// TIA Portal V16 export
// export: Created 2025-05-30T16:35:57.2781598Z, ExportSetting WithDefaults, DisplayName Totally Integrated Automation Portal, DisplayVersion V16, DisplayName TIA Portal Version Control Interface, DisplayVersion V16, DisplayName TIA Portal Openness, DisplayVersion V16, DisplayName STEP 7 Professional, DisplayVersion V16, DisplayName STEP 7 Safety, DisplayVersion V16, DisplayName WinCC Advanced, DisplayVersion V16
FUNCTION_BLOCK "Programma 1 - Test"   // FB12, GRAPH
VERSION : 0.1
// stored: AcknowledgeErrorsRequired true, AutoNumber true, CreateMinimizedDB false, IsIECCheckEnabled false, LanguageInNetworks LAD, LockOperatingMode false, PermanentILProcessingInMANMode false, SkipSteps false, UDAEnableTagReadback false, WithAlarmHandling true
   VAR_INPUT
      OFF_SQ { ExternalAccessible := 'False'; ExternalVisible := 'False'; ExternalWritable := 'False'} : Bool := false;   // Turn sequence off
      INIT_SQ { ExternalAccessible := 'False'; ExternalVisible := 'False'; ExternalWritable := 'False'} : Bool := false;   // Set sequence to initial state
      ACK_EF { ExternalAccessible := 'False'; ExternalVisible := 'False'; ExternalWritable := 'False'} : Bool := false;   // Acknowledge all errors and faults
      S_PREV { ExternalAccessible := 'False'; ExternalVisible := 'False'; ExternalWritable := 'False'} : Bool := false;   // Output previous step in parameter S_NO
      S_NEXT { ExternalAccessible := 'False'; ExternalVisible := 'False'; ExternalWritable := 'False'} : Bool := false;   // Indicate next step in parameter S_NO
      SW_AUTO { ExternalAccessible := 'False'; ExternalVisible := 'False'; ExternalWritable := 'False'} : Bool := false;   // Automatic mode
      SW_TAP { ExternalAccessible := 'False'; ExternalVisible := 'False'; ExternalWritable := 'False'} : Bool := false;   // Semiautomatic/switch with transition
      SW_TOP { ExternalAccessible := 'False'; ExternalVisible := 'False'; ExternalWritable := 'False'} : Bool := false;   // Semiautomatic/ignore transition
      SW_MAN { ExternalAccessible := 'False'; ExternalVisible := 'False'; ExternalWritable := 'False'} : Bool := false;   // Manual mode
      S_SEL { ExternalAccessible := 'False'; ExternalVisible := 'False'; ExternalWritable := 'False'} : Int := 0;   // Select step to be output to S_NO
      S_ON { ExternalAccessible := 'False'; ExternalVisible := 'False'; ExternalWritable := 'False'} : Bool := false;   // Activate step indicated in S_NO
      S_OFF { ExternalAccessible := 'False'; ExternalVisible := 'False'; ExternalWritable := 'False'} : Bool := false;   // Deactivate step indicated S_NO
      T_PUSH { ExternalAccessible := 'False'; ExternalVisible := 'False'; ExternalWritable := 'False'} : Bool := false;   // Enable transition to switch in semi automatic mode
      "Confimation Position 1" : Bool;
      "Confirmation Position 2" : Bool;
      "Products more than zero" : Bool;
      "Products zero" : Bool;
      "Timer 1" : Time;
   END_VAR
   VAR_OUTPUT
      S_NO { ExternalAccessible := 'False'; ExternalVisible := 'False'; ExternalWritable := 'False'} : Int := 0;   // Step number
      S_MORE { ExternalAccessible := 'False'; ExternalVisible := 'False'; ExternalWritable := 'False'} : Bool := false;   // More steps are available and can be shown in S_NO
      S_ACTIVE { ExternalAccessible := 'False'; ExternalVisible := 'False'; ExternalWritable := 'False'} : Bool := false;   // Step indicated in S_NO is active
      ERR_FLT { ExternalAccessible := 'False'; ExternalVisible := 'False'; ExternalWritable := 'False'} : Bool := false;   // Interlock or supervision group error
      AUTO_ON { ExternalAccessible := 'False'; ExternalVisible := 'False'; ExternalWritable := 'False'} : Bool := false;   // Automatic mode is active
      TAP_ON { ExternalAccessible := 'False'; ExternalVisible := 'False'; ExternalWritable := 'False'} : Bool := false;   // Semiautomatic mode/step with transition enabled
      TOP_ON { ExternalAccessible := 'False'; ExternalVisible := 'False'; ExternalWritable := 'False'} : Bool := false;   // Semiautomatic mode/ignore transition enabled
      MAN_ON { ExternalAccessible := 'False'; ExternalVisible := 'False'; ExternalWritable := 'False'} : Bool := false;   // Manual mode is active
      "Move Position 1" : Bool;
      "Move Position 2" : Bool;
   END_VAR
   VAR DB_SPECIFIC
      S_DISPLAY { ExternalAccessible := 'False'; ExternalVisible := 'False'; ExternalWritable := 'False'} : Int;   // Internal display of output parameter S_NO
      S_SEL_OLD { ExternalAccessible := 'False'; ExternalVisible := 'False'; ExternalWritable := 'False'} : Int;   // Previous value in S_SEL
      S_DISPIDX { ExternalAccessible := 'False'; ExternalVisible := 'False'; ExternalWritable := 'False'} : Byte;   // Index of the step in S_NO
      T_DISPIDX { ExternalAccessible := 'False'; ExternalVisible := 'False'; ExternalWritable := 'False'} : Byte;   // Index of the transition displayed in T_NO
      MOP { ExternalAccessible := 'False'; ExternalVisible := 'False'; ExternalWritable := 'False'} : Struct   // Mode
         AUTO { ExternalAccessible := 'False'; ExternalVisible := 'False'; ExternalWritable := 'False'} : Bool := true;   // Status: automatic mode
         MAN { ExternalAccessible := 'False'; ExternalVisible := 'False'; ExternalWritable := 'False'} : Bool := false;   // Status: manual mode
         TAP { ExternalAccessible := 'False'; ExternalVisible := 'False'; ExternalWritable := 'False'} : Bool := false;   // Status: semi automatic/switch with transition
         TOP { ExternalAccessible := 'False'; ExternalVisible := 'False'; ExternalWritable := 'False'} : Bool := false;   // Status: semi automatic/ignore transition
         ACK_S { ExternalAccessible := 'False'; ExternalVisible := 'False'; ExternalWritable := 'False'} : Bool := false;   // Request: acknowledge step at parameter S_NO
         REG_S { ExternalAccessible := 'False'; ExternalVisible := 'False'; ExternalWritable := 'False'} : Bool := false;   // Request: register step indicated in S_NO
         T_PREV { ExternalAccessible := 'False'; ExternalVisible := 'False'; ExternalWritable := 'False'} : Bool := false;   // Request: output previous valid transition in T_NO
         T_NEXT { ExternalAccessible := 'False'; ExternalVisible := 'False'; ExternalWritable := 'False'} : Bool := false;   // Request: output next valid transition in T_NO
         LOCK { ExternalAccessible := 'False'; ExternalVisible := 'False'; ExternalWritable := 'False'} : Bool := true;   // Status: interlocks activated
         SUP { ExternalAccessible := 'False'; ExternalVisible := 'False'; ExternalWritable := 'False'} : Bool := true;   // Status: supervisions activated
         ACKREQ { ExternalAccessible := 'False'; ExternalVisible := 'False'; ExternalWritable := 'False'} : Bool := true;   // Status: acknowledgment required
         SSKIP { ExternalAccessible := 'False'; ExternalVisible := 'False'; ExternalWritable := 'False'} : Bool := false;   // Status: "Skip steps" enabled
         OFF { ExternalAccessible := 'False'; ExternalVisible := 'False'; ExternalWritable := 'False'} : Bool := false;   // Request: deactivate all steps
         INIT { ExternalAccessible := 'False'; ExternalVisible := 'False'; ExternalWritable := 'False'} : Bool := true;   // Request: set sequence to initial state
         HALT { ExternalAccessible := 'False'; ExternalVisible := 'False'; ExternalWritable := 'False'} : Bool := false;   // Status: sequence halted
         TMS_HALT { ExternalAccessible := 'False'; ExternalVisible := 'False'; ExternalWritable := 'False'} : Bool := false;   // Status: all internal timers held
         OPS_ZERO { ExternalAccessible := 'False'; ExternalVisible := 'False'; ExternalWritable := 'False'} : Bool := false;   // Status: set all operands processed with N, L, D instructions to 0
         SACT_DISP { ExternalAccessible := 'False'; ExternalVisible := 'False'; ExternalWritable := 'False'} : Bool := true;   // Status: display active steps only
         SEF_DISP { ExternalAccessible := 'False'; ExternalVisible := 'False'; ExternalWritable := 'False'} : Bool := false;   // Status: display only steps with errors and disrupted steps
         SALL_DISP { ExternalAccessible := 'False'; ExternalVisible := 'False'; ExternalWritable := 'False'} : Bool := false;   // Status: display all steps
         S_PREV { ExternalAccessible := 'False'; ExternalVisible := 'False'; ExternalWritable := 'False'} : Bool := false;   // Request: output previous step to S_NO
         S_NEXT { ExternalAccessible := 'False'; ExternalVisible := 'False'; ExternalWritable := 'False'} : Bool := false;   // Request: Output next step at S_NO parameter
         S_SELOK { ExternalAccessible := 'False'; ExternalVisible := 'False'; ExternalWritable := 'False'} : Bool := false;   // Request: output step number from S_SEL to S_NO
         S_ON { ExternalAccessible := 'False'; ExternalVisible := 'False'; ExternalWritable := 'False'} : Bool := false;   // Request: activate step indicated in S_NO
         S_OFF { ExternalAccessible := 'False'; ExternalVisible := 'False'; ExternalWritable := 'False'} : Bool := false;   // Request: deactivate step at parameter S_NO
         T_PUSH { ExternalAccessible := 'False'; ExternalVisible := 'False'; ExternalWritable := 'False'} : Bool := false;   // Request: transition switching enabled
         REG { ExternalAccessible := 'False'; ExternalVisible := 'False'; ExternalWritable := 'False'} : Bool := false;   // Request: register all interlock and supervision errors
         ACK { ExternalAccessible := 'False'; ExternalVisible := 'False'; ExternalWritable := 'False'} : Bool := false;   // Request: acknowledge all interlock and supervision errors
         IL_PERM { ExternalAccessible := 'False'; ExternalVisible := 'False'; ExternalWritable := 'False'} : Bool := false;   // Status: permanent processing of all interlocks
         T_PERM { ExternalAccessible := 'False'; ExternalVisible := 'False'; ExternalWritable := 'False'} : Bool := false;   // Status: permanent processing of all transitions
         ILP_MAN { ExternalAccessible := 'False'; ExternalVisible := 'False'; ExternalWritable := 'False'} : Bool := false;   // Status: permanent processing of all interlocks in manual mode
      END_STRUCT;
      TICKS { ExternalAccessible := 'False'; ExternalVisible := 'False'; ExternalWritable := 'False'} : Struct   // Clock speeds
         DELTA { ExternalAccessible := 'False'; ExternalVisible := 'False'; ExternalWritable := 'False'} : Time := T#0ms;   // Time difference between cycles
         OLD { ExternalAccessible := 'False'; ExternalVisible := 'False'; ExternalWritable := 'False'} : Time := T#0ms;   // 10 ms clock counter value in last cycle
         NEW { ExternalAccessible := 'False'; ExternalVisible := 'False'; ExternalWritable := 'False'} : Time := T#0ms;   // 10 ms clock counter value in this cycle
      END_STRUCT;
      SQ_FLAGS { ExternalAccessible := 'False'; ExternalVisible := 'False'; ExternalWritable := 'False'} : Struct   // Sequence bit memory
         ERR_FLT { ExternalAccessible := 'False'; ExternalVisible := 'False'; ExternalWritable := 'False'} : Bool := false;   // Interlock and supervision group error
         ERROR { ExternalAccessible := 'False'; ExternalVisible := 'False'; ExternalWritable := 'False'} : Bool := false;   // Interlock group error
         FAULT { ExternalAccessible := 'False'; ExternalVisible := 'False'; ExternalWritable := 'False'} : Bool := false;   // Supervision group error
         RT_FAIL { ExternalAccessible := 'False'; ExternalVisible := 'False'; ExternalWritable := 'False'} : Bool := false;   // Runtime error
         NO_SNO { ExternalAccessible := 'False'; ExternalVisible := 'False'; ExternalWritable := 'False'} : Bool := false;   // Requested step number not found
         NF_OFL { ExternalAccessible := 'False'; ExternalVisible := 'False'; ExternalWritable := 'False'} : Bool := false;   // Overflow: too many ON or OFF requests
         SA_OFL { ExternalAccessible := 'False'; ExternalVisible := 'False'; ExternalWritable := 'False'} : Bool := false;   // Overflow: too many steps active
         TV_OFL { ExternalAccessible := 'False'; ExternalVisible := 'False'; ExternalWritable := 'False'} : Bool := false;   // Overflow: too many valid transitions
         MSG_OFL { ExternalAccessible := 'False'; ExternalVisible := 'False'; ExternalWritable := 'False'} : Bool := false;   // Overflow: not enough system resources for ALARM_S
         NO_SWI { ExternalAccessible := 'False'; ExternalVisible := 'False'; ExternalWritable := 'False'} : Bool := false;   // Do not switch in this cycle
         CYC_OP { ExternalAccessible := 'False'; ExternalVisible := 'False'; ExternalWritable := 'False'} : Bool := false;   // Cyclic execution of the sequence after initialization
         AS_MSG { ExternalAccessible := 'False'; ExternalVisible := 'False'; ExternalWritable := 'False'} : Bool := true;   // Alarms during runtime enabled or disabled by instruction
         AS_SEND { ExternalAccessible := 'False'; ExternalVisible := 'False'; ExternalWritable := 'False'} : Bool := false;   // Send alarms from WR_USMSG or only enter in diagnostics buffer
         SQ_BUSY { ExternalAccessible := 'False'; ExternalVisible := 'False'; ExternalWritable := 'False'} : Bool := false;   // Internal edge memory bit for sequence processing
         SA_BUSY { ExternalAccessible := 'False'; ExternalVisible := 'False'; ExternalWritable := 'False'} : Bool := false;   // Internal edge memory bit for sequence processing
         AS_SIG { ExternalAccessible := 'False'; ExternalVisible := 'False'; ExternalWritable := 'False'} : Bool := false;   // Edge memory bit for alarms from Alarm_S and Alarm_SQ
      END_STRUCT;
   END_VAR
BEGIN
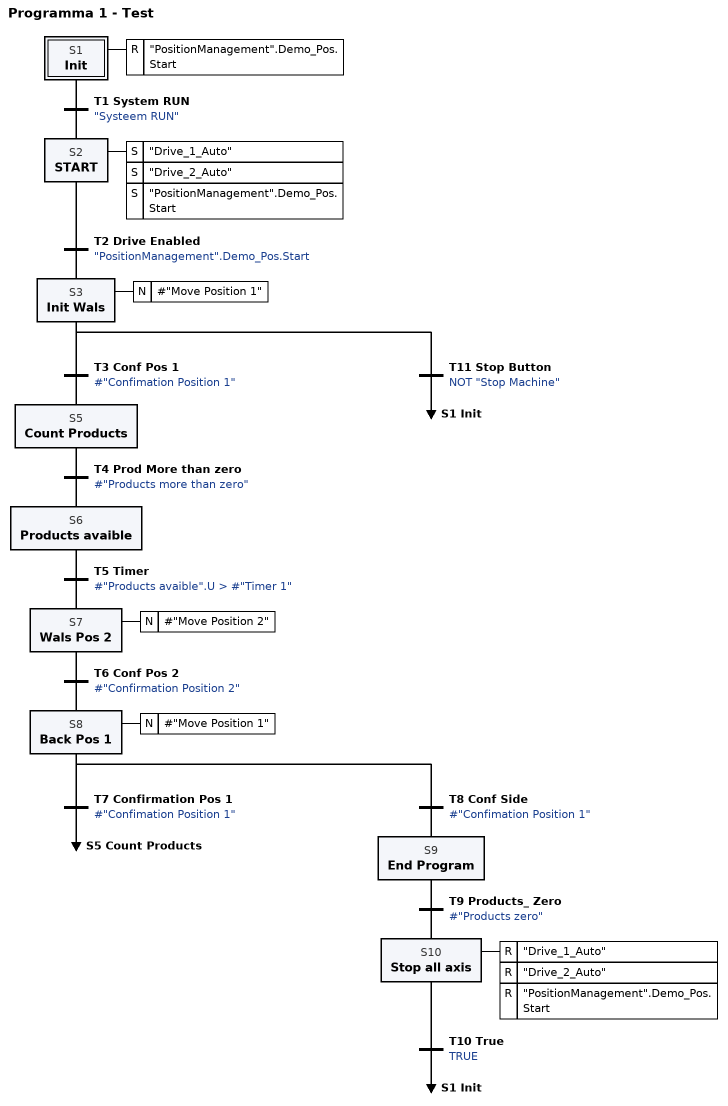
   // sequencer 1: SFC Program
   INITIAL_STEP Init:   // S1
              R    "PositionManagement".Demo_Pos.Start
   END_STEP
   TRANSITION "System RUN" FROM Init TO START   // T1
      := "Systeem RUN";
   END_TRANSITION
   STEP START:   // S2
      // Set Ouputs
              S    "Drive_1_Auto"
              S    "Drive_2_Auto"
              S    "PositionManagement".Demo_Pos.Start
   END_STEP
   TRANSITION "Drive Enabled" FROM START TO "Init Wals"   // T2
      := "PositionManagement".Demo_Pos.Start;
   END_TRANSITION
   STEP "Init Wals":   // S3
      // Move Start Position4
              N    #"Move Position 1"
   END_STEP
   TRANSITION "Conf Pos 1" FROM "Init Wals" TO "Count Products"   // T3
      := #"Confimation Position 1";
   END_TRANSITION
   TRANSITION "Stop Button" FROM "Init Wals" TO Init   // T11, jump
      := NOT "Stop Machine";
   END_TRANSITION
   STEP "Count Products":   // S5
   END_STEP
   TRANSITION "Prod More than zero" FROM "Count Products" TO "Products avaible"   // T4
      := #"Products more than zero";
   END_TRANSITION
   STEP "Products avaible":   // S6
   END_STEP
   TRANSITION "Timer" FROM "Products avaible" TO "Wals Pos 2"   // T5: Timer 1
      := #"Products avaible".U > #"Timer 1";
   END_TRANSITION
   STEP "Wals Pos 2":   // S7
              N    #"Move Position 2"
   END_STEP
   TRANSITION "Conf Pos 2" FROM "Wals Pos 2" TO "Back Pos 1"   // T6
      := #"Confirmation Position 2";
   END_TRANSITION
   STEP "Back Pos 1":   // S8
      // Move Position 1
              N    #"Move Position 1"
   END_STEP
   TRANSITION "Confirmation Pos 1" FROM "Back Pos 1" TO "Count Products"   // T7, jump: Conf Pos 1
      := #"Confimation Position 1";
   END_TRANSITION
   TRANSITION "Conf Side" FROM "Back Pos 1" TO "End Program"   // T8
      := #"Confimation Position 1";
   END_TRANSITION
   STEP "End Program":   // S9
   END_STEP
   TRANSITION "Products_ Zero" FROM "End Program" TO "Stop all axis"   // T9
      := #"Products zero";
   END_TRANSITION
   STEP "Stop all axis":   // S10
      // Reset Axis
              R    "Drive_1_Auto"
              R    "Drive_2_Auto"
              R    "PositionManagement".Demo_Pos.Start
   END_STEP
   TRANSITION True FROM "Stop all axis" TO Init   // T10, jump
      := TRUE;
   END_TRANSITION
END_FUNCTION_BLOCK
